// TIA Portal V17 export
// export: Created 2025-06-26T07:49:50.9138359Z, ExportSetting WithDefaults, DisplayName Totally Integrated Automation Portal, DisplayVersion V17 Update 8, DisplayName TIA Portal Openness, DisplayVersion V17 Update 8, DisplayName TIA Portal Version Control Interface, DisplayVersion V17, DisplayName STEP 7 Professional, DisplayVersion V17 Update 8, DisplayName STEP 7 Safety, DisplayVersion V17 Update 6, DisplayName WinCC Advanced, DisplayVersion V17 Update 8
DATA_BLOCK "DB_Profiling"   // DB100
{ S7_Optimized_Access := 'TRUE' }
AUTHOR : Heaten
VERSION : 0.1
// stored: AutoNumber false, DBAccessibleFromOPCUA true, DBAccessibleFromWebserver true, IsOnlyStoredInLoadMemory false, IsRetainMemResEnabled false, IsWriteProtectedInAS false, MemoryReserve 100
   VAR
      OB1time : "stProfile";
      OB30time { S7_SetPoint := 'True'} : "stProfile";
      Section10time : "stProfile";
      Section20time : "stProfile";
      Section30time : "stProfile";
      Section40time : "stProfile";
      Section60time : "stProfile";
      Section80time : "stProfile";
      Section90time : "stProfile";
      Section10_DigitalInputProcessing { S7_SetPoint := 'True'} : "stProfile";
      Section10_AnalogInputProcessing { S7_SetPoint := 'True'} : "stProfile";
      Section10_InverterDriveProcessing { S7_SetPoint := 'True'} : "stProfile";
      Section10_InputAlarmHandling { S7_SetPoint := 'True'} : "stProfile";
      Section20_Calculations { S7_SetPoint := 'True'} : "stProfile";
      Section20_StateMachine { S7_SetPoint := 'True'} : "stProfile";
      Section20_ControlAlarmHandling { S7_SetPoint := 'True'} : "stProfile";
      Section20_Regulation { S7_SetPoint := 'True'} : "stProfile";
      Section20_StartStopControl { S7_SetPoint := 'True'} : "stProfile";
   END_VAR
BEGIN
END_DATA_BLOCK
